Staubli VAL3: WeldAction.pgx

public program WeldAction()
begin

  //焊接收弧点
  dDio["UsO_bNull5"]=true
  // delay(0.005)
  call Digtal2AnalogS(0)



end
